// TIA Portal V16 export
// export: Created 2021-11-12T13:32:29.7923349Z, ExportSetting WithDefaults, DisplayName Totally Integrated Automation Portal, DisplayVersion V16 Update 3, DisplayName TIA Portal Version Control Interface, DisplayVersion V16 Update 2, DisplayName TIA Portal Openness, DisplayVersion V16 Update 3, DisplayName SINAMICS Startdrive Advanced, DisplayVersion V16 Update 5, DisplayName SINAMICS Startdrive G130, G150, S120, S150, SINAMICS MV, S210, DisplayVersion V16 Update 5, DisplayName SINAMICS Startdrive G110M, G120, G120C, G120D, G120P, G115D, DisplayVersion V16 Update 5, DisplayName STEP 7 Professional, DisplayVersion V16 Update 3, DisplayName STEP 7 Safety, DisplayVersion V16, DisplayName WinCC UA Professional, DisplayVersion V16 Update 3
DATA_BLOCK "HMI_CMD_1R3"   // DB140
{ S7_Optimized_Access := 'TRUE' }
VERSION : 0.1
// stored: AutoNumber true, DBAccessibleFromOPCUA true, IsOnlyStoredInLoadMemory false, IsRetainMemResEnabled false, IsWriteProtectedInAS false, MemoryReserve 100
   VAR
      xxxxx___BinarySensors___xxxxx_1 : Byte;
      "CL01-BG01_4" { S7_SetPoint := 'True'} : "UDT_CH_DI_Command";   // Robot 1R3 Gripper on table 1
      "CL02-BG01_4" { S7_SetPoint := 'True'} : "UDT_CH_DI_Command";   // Robot 1R3 Gripper on table 2
      "RO01-BG10_2" { S7_SetPoint := 'True'} : "UDT_CH_DI_Command";   // Robot 1R3 senzor piston lubrication printed / Robot 1R3 senzor pístu mazivo vytlačeno
      xxxxx___BinaryOthers___xxxxx_1 : Byte;
      PwrOK : "UDT_CH_DI_Command";
      "100+UF01-SF02_12" { S7_SetPoint := 'True'} : "UDT_CH_DI_Command";   // Robot 1R3, 1R4 immediate stop
      "000+UH10-SF26_12" { S7_SetPoint := 'True'} : "UDT_CH_DI_Command";   // Okamžitý stop Robot 1R3, 1R4
      xxxxx___AnalogueSensors___xxxxx_1 : Byte;
      xxxxx___Drives___xxxxx_1 : Byte;
      RO01 : "UDT_RobotABB_Command";   // Robot
      RC01 : "UDT_DriveRobotABB_Command";   // Controller
      Gripper : "UDT_RobotGripper_Command";   // Gripper
      ParkPosReq : Bool;   // Go to parking position
      xxxxx___Others___xxxxx_1 : Byte;
      MatCard : "UDT_MatCard_Cmd";   // Material card commands
      Sequence : "UDT_Sequence_Command";
      xxxxx___SensorAlarms___xxxxx : Byte;
      RO01_Timeout : "UDT_DI_Mon_Command";   // Robot job active for too long
      CL01_BG01 { S7_SetPoint := 'True'} : "UDT_DI_Mon_Command";   // gripper on upper table
      CL01_BG02 { S7_SetPoint := 'True'} : "UDT_DI_Mon_Command";   // gripper on lower table
      ES { S7_SetPoint := 'True'} : "UDT_DI_Mon_Command";   // E-stop
      "RO01-BG10" { S7_SetPoint := 'True'} : "UDT_DI_Mon_Command";   // Robot 1R3 senzor piston lubrication not printed / Robot 1R3 senzor pístu mazivo nevytlačeno
   END_VAR
BEGIN
END_DATA_BLOCK
